// Mitsubishi GX Works2 project: z07   PLC: Q02/Q02H

PROGRAM MAIN
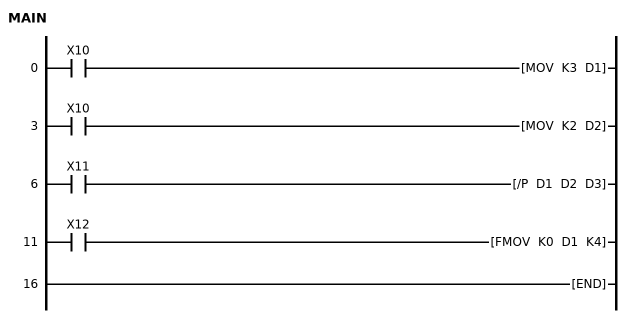
0     LD      X10
      MOV     K3 D1
3     LD      X10
      MOV     K2 D2
6     LD      X11
      /P      D1 D2 D3
11    LD      X12
      FMOV    K0 D1 K4
16    END
END_PROGRAM
